{attribute addProperty BoxType "EL3001-0000-0016"}
{attribute addProperty Id "AI_StandardAT %I*AI_Standard_BC62E3BB7290WcStateAT %I*WcState_98A4DF7520.250InfoDataAT %I*InfoData_BC63D37F80100"}
{attribute addProperty CRC "2077206891"}
{attribute addProperty SizeInBites "154"}
{attribute addProperty SizeInBytes "19.25"}
TYPE EL3001_14E7B212 :
STRUCT
	{attribute addProperty Name "AI_Standard"}
	AI_Standard : AI_Standard_BC62E3BB;
	{attribute addProperty Name "WcState"}
	WcState : WcState_98A4DF75;
	{attribute addProperty Name "InfoData"}
	InfoData : InfoData_BC63D37F;
END_STRUCT
END_TYPE

(* stored: Version 1.2.0.0, ProductVersion 3.1.4024.9
   DUT EL3001_14E7B212: Id {d87b156c-b044-4bdc-8450-2231c61b1fe9} *)
